# EPICS substitutions: iocBoot/ioc13MeasComp2408_1/USB2408.substitutions
file "$(MEASCOMP)/measCompApp/Db/measCompLongIn.template"
{
pattern
{              P,   R,   MASK,       PORT,  ADDR}
{   13USB2408_1:,  Li,   0xFF,  USB2408_1,     0}
}

file "$(MEASCOMP)/measCompApp/Db/measCompBinaryIn.template"
{
pattern
{              P,    R,  MASK,        PORT,  ADDR}
{   13USB2408_1:,  Bi1,  0x01,   USB2408_1,     0}
{   13USB2408_1:,  Bi2,  0x02,   USB2408_1,     0}
{   13USB2408_1:,  Bi3,  0x04,   USB2408_1,     0}
{   13USB2408_1:,  Bi4,  0x08,   USB2408_1,     0}
{   13USB2408_1:,  Bi5,  0x10,   USB2408_1,     0}
{   13USB2408_1:,  Bi6,  0x20,   USB2408_1,     0}
{   13USB2408_1:,  Bi7,  0x40,   USB2408_1,     0}
{   13USB2408_1:,  Bi8,  0x80,   USB2408_1,     0}
}

file "$(MEASCOMP)/measCompApp/Db/measCompLongOut.template"
{
pattern
{              P,   R,   MASK,       PORT,  ADDR}
{   13USB2408_1:,  Lo,   0xFF,  USB2408_1,     0}
}

file "$(MEASCOMP)/measCompApp/Db/measCompBinaryOut.template"
{
pattern
{              P,    R,  MASK,        PORT,  ADDR}
{   13USB2408_1:,  Bo1,  0x01,   USB2408_1,     0}
{   13USB2408_1:,  Bo2,  0x02,   USB2408_1,     0}
{   13USB2408_1:,  Bo3,  0x04,   USB2408_1,     0}
{   13USB2408_1:,  Bo4,  0x08,   USB2408_1,     0}
{   13USB2408_1:,  Bo5,  0x10,   USB2408_1,     0}
{   13USB2408_1:,  Bo6,  0x20,   USB2408_1,     0}
{   13USB2408_1:,  Bo7,  0x40,   USB2408_1,     0}
{   13USB2408_1:,  Bo8,  0x80,   USB2408_1,     0}
}

# Direction bits on binary I/O
#  VAL 0=input, 1=output
file "$(MEASCOMP)/measCompApp/Db/measCompBinaryDir.template"
{
pattern
{              P,    R,  MASK,  VAL,       PORT,  ADDR}
{   13USB2408_1:,  Bd1,  0x01,    0,  USB2408_1,     0}
{   13USB2408_1:,  Bd2,  0x02,    0,  USB2408_1,     0}
{   13USB2408_1:,  Bd3,  0x04,    0,  USB2408_1,     0}
{   13USB2408_1:,  Bd4,  0x08,    0,  USB2408_1,     0}
{   13USB2408_1:,  Bd5,  0x10     1,  USB2408_1,     0}
{   13USB2408_1:,  Bd6,  0x20,    1,  USB2408_1,     0}
{   13USB2408_1:,  Bd7,  0x40,    1,  USB2408_1,     0}
{   13USB2408_1:,  Bd8,  0x80,    1,  USB2408_1,     0}
}

file "$(MEASCOMP)/measCompApp/Db/1608GCounter.template"
{
pattern
{              P,         R,       PORT,   ADDR}
{   13USB2408_1:,  Counter1,  USB2408_1,      0}
{   13USB2408_1:,  Counter2,  USB2408_1,      1}
}

# Analog inputs
file "$(MEASCOMP)/measCompApp/Db/measCompAnalogIn.template"
{
pattern
{              P,     R,      PORT, ADDR,  EGUL, LOPR, EGUF, HOPR, RANGE,       SCAN, PREC}
{   13USB2408_1:,   Ai1, USB2408_1,    0,  -10., -10.,  10.,  10.,    3,  "1 second",   4}
{   13USB2408_1:,   Ai2, USB2408_1,    1,  -10., -10.,  10.,  10.,    3,  "1 second",   4}
{   13USB2408_1:,   Ai3, USB2408_1,    2,   -5.,  -5.,   5.,   5.,    2,  "1 second",   4}
{   13USB2408_1:,   Ai4, USB2408_1,    3,   -5.,  -5.,   5.,   5.,    2,  "1 second",   4}
{   13USB2408_1:,   Ai5, USB2408_1,    4,   -2.,  -2.,   2.,   2.,    1,  "1 second",   4}
{   13USB2408_1:,   Ai6, USB2408_1,    5,   -2.,  -2.,   2.,   2.,    1,  "1 second",   4}
{   13USB2408_1:,   Ai7, USB2408_1,    6,   -1.,  -1.,   1.,   1.,    0,  "1 second",   4}
{   13USB2408_1:,   Ai8, USB2408_1,    7,   -1.,  -1.,   1.,   1.,    0,  "1 second",   4}
}

# Temperature inputs
file "$(MEASCOMP)/measCompApp/Db/measCompTemperatureIn.template"
{
pattern
{              P,     R,      PORT, ADDR,       SCAN, PREC}
{   13USB2408_1:,   Ti1, USB2408_1,    0, "1 second",   2}
{   13USB2408_1:,   Ti2, USB2408_1,    1, "1 second",   2}
{   13USB2408_1:,   Ti3, USB2408_1,    2, "1 second",   2}
{   13USB2408_1:,   Ti4, USB2408_1,    3, "1 second",   2}
{   13USB2408_1:,   Ti5, USB2408_1,    4, "1 second",   2}
{   13USB2408_1:,   Ti6, USB2408_1,    5, "1 second",   2}
{   13USB2408_1:,   Ti7, USB2408_1,    6, "1 second",   2}
{   13USB2408_1:,   Ti8, USB2408_1,    7, "1 second",   2}
}

# Waveform digitzer
file "$(MEASCOMP)/measCompApp/Db/measCompWaveformDig.template"
{
pattern
{              P,        R,         PORT,  ADDR, MAX_POINTS,    PREC}
{   13USB2408_1:,  WaveDig,    USB2408_1,     0,       2048,       4}
}

file "$(MEASCOMP)/measCompApp/Db/measCompWaveformDigN.template"
{
pattern
{              P,         R,        PORT,  ADDR, MAX_POINTS,    PREC}
{   13USB2408_1:,  WaveDig1,   USB2408_1,     0,       2048,       4}
{   13USB2408_1:,  WaveDig2,   USB2408_1,     1,       2048,       4}
{   13USB2408_1:,  WaveDig3,   USB2408_1,     2,       2048,       4}
{   13USB2408_1:,  WaveDig4,   USB2408_1,     3,       2048,       4}
{   13USB2408_1:,  WaveDig5,   USB2408_1,     4,       2048,       4}
{   13USB2408_1:,  WaveDig6,   USB2408_1,     5,       2048,       4}
{   13USB2408_1:,  WaveDig7,   USB2408_1,     6,       2048,       4}
{   13USB2408_1:,  WaveDig8,   USB2408_1,     7,       2048,       4}
}

# Analog outputs
file "$(MEASCOMP)/measCompApp/Db/measCompAnalogOut.template"
{
pattern
{              P,    R, VAL,       PORT, ADDR,  EGUL, DRVL, LOPR, EGUF, DRVH, HOPR, PREC}
{   13USB2408_1:,  Ao1,   0,  USB2408_1,    0,  -10., -10., -10.,  10.,  10.,  10.,    4}
{   13USB2408_1:,  Ao2,   0,  USB2408_1,    1,  -10., -10., -10.,  10.,  10.,  10.,    4}
}

# Waveform generator
file "$(MEASCOMP)/measCompApp/Db/measCompWaveformGen.template"
{
pattern
{              P,        R,         PORT,  ADDR, MAX_POINTS,    PREC}
{   13USB2408_1:,  WaveGen,    USB2408_1,     0,      2048,        4}
}
file "$(MEASCOMP)/measCompApp/Db/measCompWaveformGenN.template"
{
pattern
{              P,         R,        PORT,  ADDR, MAX_POINTS,    PREC}
{   13USB2408_1:,  WaveGen1,   USB2408_1,     0,      2048,        4}
{   13USB2408_1:,  WaveGen2,   USB2408_1,     1,      2048,        4}
}
